// TIA Portal V17 export
// export: Created 2025-06-25T13:13:11.2991386Z, ExportSetting WithDefaults, DisplayName Totally Integrated Automation Portal, DisplayVersion V17 Update 8, DisplayName TIA Portal Openness, DisplayVersion V17 Update 8, DisplayName TIA Portal Version Control Interface, DisplayVersion V17, DisplayName STEP 7 Professional, DisplayVersion V17 Update 8, DisplayName STEP 7 Safety, DisplayVersion V17 Update 6, DisplayName WinCC Advanced, DisplayVersion V17 Update 8
FUNCTION "State7_Stop" : Void   // FC57, FBD
{ S7_Optimized_Access := 'TRUE' }
VERSION : 0.1
// stored: AutoNumber true, IsIECCheckEnabled false, SetENOAutomatically false, UDAEnableTagReadback false
   VAR_INPUT
      Active : Bool;
   END_VAR
   VAR_OUTPUT
      Offline : Bool;
   END_VAR
BEGIN

REGION Network 1: State number
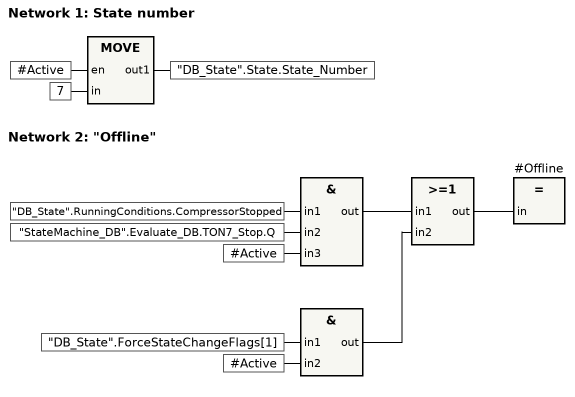
   IF #Active THEN "DB_State".State.State_Number := 7; END_IF;
END_REGION

REGION Network 2: "Offline"
   #Offline := ("DB_State".RunningConditions.CompressorStopped AND "StateMachine_DB".Evaluate_DB.TON7_Stop.Q AND #Active) OR ("DB_State".ForceStateChangeFlags[1] AND #Active);
END_REGION
END_FUNCTION
